FUNCTION_BLOCK PiperNullContext IMPLEMENTS IPluginRunner

METHOD RegisterPlugin
VAR_INPUT
	plugin : IPlugin;
END_VAR
END_METHOD

END_FUNCTION_BLOCK

(* stored: Version 1.1.0.1, ProductVersion 3.1.4024.12
   POU PiperNullContext: Id {07930393-8d34-430f-86f6-cac95646cb0a}, SpecialFunc None
   Method RegisterPlugin: Id {f95b39e0-6a5d-473e-a936-153bf944be5b} *)
